FUNCTION_BLOCK PUBLIC ABSTRACT TcoTixonFeedingTask EXTENDS TcoCore.TcoTask
VAR
    _errorMessage : TcoCore.TcoMessenger(THIS^);
    {attribute 'hide'}
    _progress : INT := 0;
    {attribute 'hide'}
    _infoTimer : TON;
    _infoTime : TIME;
    {attribute 'hide'}
    _errorTimer : TON;
    _errorTime : TIME;
    {attribute 'hide'}
    _timer : TON;
    {attribute 'hide'}
    _varInfo : __SYSTEM.VAR_INFO;
    {attribute 'hide'}
    _sb : TcoCore.StringBuilder;
    {attribute 'hide'}
    _autoRestore : BOOL;
END_VAR

PROPERTY PUBLIC AutoRestore : BOOL
GET
AutoRestore := _autoRestore;
END_GET
SET
_autoRestore := AutoRestore;
END_SET
END_PROPERTY

METHOD CallTimers
VAR_INPUT
    inValue : BOOL;
END_VAR
IF THIS^.ErrorTime <> T#0S OR NOT inValue THEN
    _errorTimer(IN := inValue, PT := THIS^.ErrorTime);
END_IF;

IF THIS^.InfoTime <> T#0S OR NOT inValue THEN
    _infoTimer(IN := inValue, PT := THIS^.InfoTime);
END_IF;
END_METHOD

PROPERTY PUBLIC ErrorTime : REFERENCE TO TIME
GET
ErrorTime REF= _errorTime;
END_GET
END_PROPERTY

PROPERTY InfoTime : REFERENCE TO TIME
GET
InfoTime REF= _infoTime;
END_GET
END_PROPERTY

(*~
    <docu>
        <summary>
            Restores this instance to the Ready state. Can be called explicitly or from within one of the restore mechanisms.
            <para>
                See also <see cref="PlcDocu.TcoCore.TcoTask.AutoRestorable()"/>
            </para>
        </summary>
    </docu>
~*)
METHOD Restore : ITcoRestorable
SUPER^.Restore();
_progress := 0;
_timer(In := FALSE);
CallTimers(FALSE);
Messenger.UnPin();
_errorMessage.UnPin();
_autoRestore := false;
END_METHOD

END_FUNCTION_BLOCK

(* stored: Version 1.1.0.1, ProductVersion 3.1.4024.12
   POU TcoTixonFeedingTask: Id {3c2fc736-bc66-08d9-20ec-4296aae9c0c4}, SpecialFunc None
   Property AutoRestore: Id {b2c74594-a4f6-05fc-1e25-48d1cf294532}
   Get Get: Id {efd33750-311a-075a-3a08-942e3ab53a2c}
   Set Set: Id {df96d8c9-1856-0e3a-2f28-997fd0542776}
   Method CallTimers: Id {ecb7089a-a7b9-01c1-1e99-ab26e8329008}
   Property ErrorTime: Id {9a36ad8c-8f87-0010-18f2-6a40d936c74f}
   Get Get: Id {50db764d-a7e6-07f2-3b4c-3620466826ea}
   Property InfoTime: Id {2c67b3aa-4958-0588-0780-e699e5aa3de9}
   Get Get: Id {0fcfb362-3ecc-0c97-0b84-c5e2d531cd4c}
   Method Restore: Id {ad9a6d70-9aaa-0604-0057-a45c21976679} *)
